LIN {X 0,Y 31.532,Z 556.108,A -85,B 0,C 180,E1 -28751.981,E2 -28751.981} C_VEL
LIN {X 0,Y 25.561,Z 556.328,A -85,B 0,C 180,E1 -28725.977,E2 -28725.977} C_VEL
LIN {X 0,Y 24.732,Z 555.913,A -85,B 0,C 180,E1 -28710.018,E2 -28710.018} C_VEL
LIN {X 0,Y 28.547,Z 553.832,A -85,B 0,C 180,E1 -28680.521,E2 -28680.521} C_VEL
LIN {X 0,Y 35.086,Z 551.171,A -85,B 0,C 180,E1 -28665.504,E2 -28665.504} C_VEL
LIN {X 0,Y 43.077,Z 547.529,A -85,B 0,C 180,E1 -28655.356,E2 -28655.356} C_VEL
LIN {X 0,Y 45.151,Z 546.482,A -85,B 0,C 180,E1 -28653.412,E2 -28653.412} C_VEL
LIN {X 0,Y 49.316,Z 544.218,A -85,B 0,C 180,E1 -28649.112,E2 -28649.112} C_VEL
LIN {X 0,Y 55.529,Z 540.262,A -85,B 0,C 180,E1 -28641.789,E2 -28641.789} C_VEL
LIN {X 0,Y 62.09,Z 535.634,A -85,B 0,C 180,E1 -28636.105,E2 -28636.105} C_VEL
LIN {X 0,Y 66.48,Z 532.294,A -85,B 0,C 180,E1 -28634.227,E2 -28634.227} C_VEL
LIN {X 0,Y 72.039,Z 527.678,A -85,B 0,C 180,E1 -28632.719,E2 -28632.719} C_VEL
LIN {X 0,Y 72.567,Z 527.178,A -85,B 0,C 180,E1 -28631.17,E2 -28631.17} C_VEL
LIN {X 0,Y 73.811,Z 526.27,A -85,B 0,C 180,E1 -28625.465,E2 -28625.465} C_VEL
LIN {X 0,Y 73.778,Z 526.492,A -85,B 0,C 180,E1 -28623.847,E2 -28623.847} C_VEL
LIN {X 0,Y 72.977,Z 527.348,A -85,B 0,C 180,E1 -28623.003,E2 -28623.003} C_VEL
LIN {X 0,Y 62.759,Z 536.223,A -85,B 0,C 180,E1 -28620.002,E2 -28620.002} C_VEL
LIN {X 0,Y 52.835,Z 543.411,A -85,B 0,C 180,E1 -28615.924,E2 -28615.924} C_VEL
LIN {X 0,Y 46.098,Z 547.609,A -85,B 0,C 180,E1 -28612.222,E2 -28612.222} C_VEL
LIN {X 0,Y 36.085,Z 552.615,A -85,B 0,C 180,E1 -28606.803,E2 -28606.803} C_VEL
LIN {X 0,Y 26.676,Z 556.503,A -85,B 0,C 180,E1 -28597.191,E2 -28597.191} C_VEL
LIN {X 0,Y 18.844,Z 559.379,A -85,B 0,C 180,E1 -28578.201,E2 -28578.201} C_VEL
LIN {X 0,Y 15.71,Z 560.785,A -85,B 0,C 180,E1 -28556.543,E2 -28556.543} C_VEL
LIN {X 0,Y 15.516,Z 561.743,A -85,B 0,C 180,E1 -28529.972,E2 -28529.972} C_VEL
LIN {X 0,Y 16.776,Z 561.911,A -85,B 0,C 180,E1 -28496.905,E2 -28496.905} C_VEL
LIN {X 0,Y 24.129,Z 561.067,A -85,B 0,C 180,E1 -28469.059,E2 -28469.059} C_VEL
LIN {X 0,Y 26.701,Z 560.294,A -85,B 0,C 180,E1 -28460.55,E2 -28460.55} C_VEL
LIN {X 0,Y 31.609,Z 556.596,A -85,B 0,C 180,E1 -28413.593,E2 -28413.593} C_VEL
LIN {X 0,Y 32.391,Z 556.347,A -85,B 0,C 180,E1 -28410.239,E2 -28410.239} C_VEL
LIN {X 0,Y 26.722,Z 557.1,A -85,B 0,C 180,E1 -28402.12,E2 -28402.12} C_VEL
LIN {X 0,Y 18.902,Z 557.337,A -85,B 0,C 180,E1 -28371.852,E2 -28371.852} C_VEL
LIN {X 0,Y 17.703,Z 556.934,A -85,B 0,C 180,E1 -28350.025,E2 -28350.025} C_VEL
LIN {X 0,Y 22.713,Z 554.871,A -85,B 0,C 180,E1 -28311.792,E2 -28311.792} C_VEL
LIN {X 0,Y 30.477,Z 552.23,A -85,B 0,C 180,E1 -28296.211,E2 -28296.211} C_VEL
LIN {X 0,Y 39.436,Z 548.606,A -85,B 0,C 180,E1 -28287.017,E2 -28287.017} C_VEL
LIN {X 0,Y 48.918,Z 543.9,A -85,B 0,C 180,E1 -28280.983,E2 -28280.983} C_VEL
LIN {X 0,Y 58.688,Z 537.968,A -85,B 0,C 180,E1 -28276.689,E2 -28276.689} C_VEL
LIN {X 0,Y 66.48,Z 532.294,A -85,B 0,C 180,E1 -28274.227,E2 -28274.227} C_VEL
LIN {X 0,Y 66.615,Z 532.173,A -85,B 0,C 180,E1 -28273.414,E2 -28273.414} C_VEL
LIN {X 0,Y 65.377,Z 533.124,A -85,B 0,C 180,E1 -28271.686,E2 -28271.686} C_VEL
LIN {X 0,Y 61.341,Z 536.219,A -85,B 0,C 180,E1 -28268.901,E2 -28268.901} C_VEL
LIN {X 0,Y 51.92,Z 542.722,A -85,B 0,C 180,E1 -28264.379,E2 -28264.379} C_VEL
LIN {X 0,Y 44.976,Z 546.829,A -85,B 0,C 180,E1 -28261.36,E2 -28261.36} C_VEL
LIN {X 0,Y 42.554,Z 548.097,A -85,B 0,C 180,E1 -28260.535,E2 -28260.535} C_VEL
LIN {X 0,Y 31.665,Z 552.937,A -85,B 0,C 180,E1 -28256.869,E2 -28256.869} C_VEL
LIN {X 0,Y 21.428,Z 556.495,A -85,B 0,C 180,E1 -28249.603,E2 -28249.603} C_VEL
LIN {X 0,Y 9.811,Z 559.726,A -85,B 0,C 180,E1 -28215.689,E2 -28215.689} C_VEL
LIN {X 0,Y 8.334,Z 560.704,A -85,B 0,C 180,E1 -28169.948,E2 -28169.948} C_VEL
LIN {X 0,Y 11.117,Z 560.892,A -85,B 0,C 180,E1 -28119.199,E2 -28119.199} C_VEL
LIN {X 0,Y 17.272,Z 560.523,A -85,B 0,C 180,E1 -28098.447,E2 -28098.447} C_VEL
LIN {X 0,Y 19.011,Z 560.193,A -85,B 0,C 180,E1 -28092.824,E2 -28092.824} C_VEL
LIN {X 0,Y 22.001,Z 558.293,A -85,B 0,C 180,E1 -28057.785,E2 -28057.785} C_VEL
LIN {X 0,Y 20.969,Z 558.235,A -85,B 0,C 180,E1 -28052.732,E2 -28052.732} C_VEL
LIN {X 0,Y 12.651,Z 558.346,A -85,B 0,C 180,E1 -28023.787,E2 -28023.787} C_VEL
LIN {X 0,Y 10.675,Z 557.953,A -85,B 0,C 180,E1 -27990.041,E2 -27990.041} C_VEL
LIN {X 0,Y 12.851,Z 557.135,A -85,B 0,C 180,E1 -27956.887,E2 -27956.887} C_VEL
LIN {X 0,Y 23.73,Z 554.288,A -85,B 0,C 180,E1 -27927.358,E2 -27927.358} C_VEL
LIN {X 0,Y 33.465,Z 551.008,A -85,B 0,C 180,E1 -27919.124,E2 -27919.124} C_VEL
LIN {X 0,Y 43.474,Z 546.71,A -85,B 0,C 180,E1 -27914.122,E2 -27914.122} C_VEL
LIN {X 0,Y 55.374,Z 540.153,A -85,B 0,C 180,E1 -27910.434,E2 -27910.434} C_VEL
LIN {X 0,Y 63.934,Z 534.335,A -85,B 0,C 180,E1 -27908.426,E2 -27908.426} C_VEL
LIN {X 0,Y 63.717,Z 534.597,A -85,B 0,C 180,E1 -27906.988,E2 -27906.988} C_VEL
LIN {X 0,Y 52.842,Z 542.214,A -85,B 0,C 180,E1 -27904.171,E2 -27904.171} C_VEL
LIN {X 0,Y 45.688,Z 546.458,A -85,B 0,C 180,E1 -27901.423,E2 -27901.423} C_VEL
LIN {X 0,Y 42.554,Z 548.097,A -85,B 0,C 180,E1 -27900.535,E2 -27900.535} C_VEL
LIN {X 0,Y 36.947,Z 550.696,A -85,B 0,C 180,E1 -27899.743,E2 -27899.743} C_VEL
LIN {X 0,Y 31.094,Z 552.85,A -85,B 0,C 180,E1 -27900.494,E2 -27900.494} C_VEL
LIN {X 0,Y 19.127,Z 556.163,A -85,B 0,C 180,E1 -27905.162,E2 -27905.162} C_VEL
LIN {X 0,Y 13.043,Z 557.508,A -85,B 0,C 180,E1 -27906.825,E2 -27906.825} C_VEL
LIN {X 0,Y 11.007,Z 557.869,A -85,B 0,C 180,E1 -27906.302,E2 -27906.302} C_VEL
LIN {X 0,Y 1.154,Z 559.665,A -85,B 0,C 180,E1 -27809.621,E2 -27809.621} C_VEL
LIN {X 0,Y 7.921,Z 559.871,A -85,B 0,C 180,E1 -27719.987,E2 -27719.987} C_VEL
LIN {X 0,Y 12.38,Z 559.626,A -85,B 0,C 180,E1 -27711.904,E2 -27711.904} C_VEL
LIN {X 0,Y 7.852,Z 559.354,A -85,B 0,C 180,E1 -27693.647,E2 -27693.647} C_VEL
LIN {X 0,Y 3.647,Z 558.971,A -85,B 0,C 180,E1 -27630.12,E2 -27630.12} C_VEL
LIN {X 0,Y 7.953,Z 558.168,A -85,B 0,C 180,E1 -27568.029,E2 -27568.029} C_VEL
LIN {X 0,Y 21.43,Z 555.338,A -85,B 0,C 180,E1 -27550.425,E2 -27550.425} C_VEL
LIN {X 0,Y 21.342,Z 555.416,A -85,B 0,C 180,E1 -27549.047,E2 -27549.047} C_VEL
LIN {X 0,Y 11.007,Z 557.869,A -85,B 0,C 180,E1 -27546.302,E2 -27546.302} C_VEL
LIN {X 0,Y 9.406,Z 559.831,A -85,B 0,C 180,E1 -27545.303,E2 -27545.303} C_VEL
LIN {X 0,Y 9.406,Z 600,A -85,B 0,C 180,E1 -27545.303,E2 -27545.303} C_VEL
LIN {X 0,Y 9.406,Z 600,A -85,B 0,C 180,E1 -27545.303,E2 -27545.303}

QRS_NEXT_CUT()

QRS_NEXT()
QRS_HOME()

END
